Universal Robots PolyScope program: cubeDev.urp

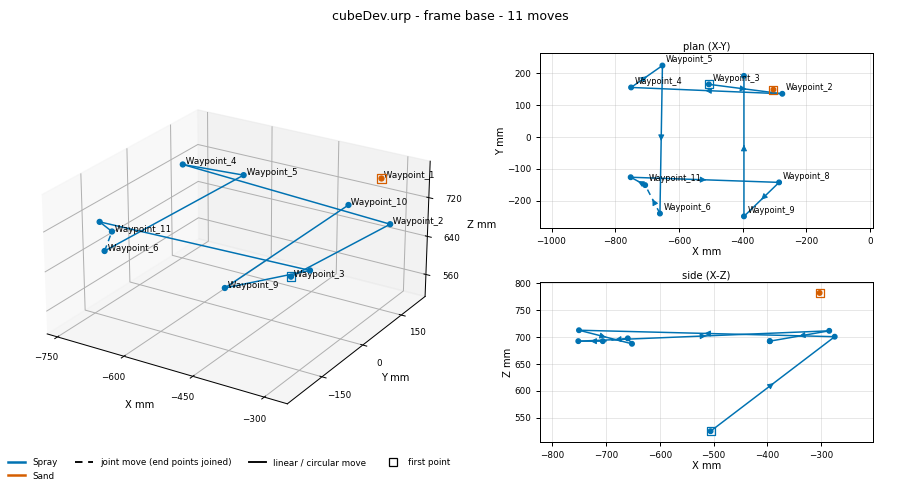
[picture p0: tool path of cubeDev.urp in frame base, 11 of 11 moves have a stored position in this frame; points joined in program order, loops and branches not executed]
Program cubeDev (installation=CubeDev directory=/programs/cube/archive createdIn=5.11.5.1010327 lastSavedIn=5.11.5.1010327 robotSerialNumber=20215500677)
Calibrated DH parameters: a=[0.000204, -0.239222, -0.391845, -0.000001, 0.000022, 0]; d=[0.162722, -355.808559, 353.37206, 2.570385, 0.099741, 0.099629]; alpha=[1.571124, 0.000988, 0.008295, 1.568963, -1.570303, 0]; deltaTheta=[0, -0.973091, 7.204745, 0.05153, 0, 0]
Robot Program (runOnlyOnce=false)
  Wait Sleep waitTime=0.01
SuppressedNode
  SubProgram LoadCube (keepSynchronizedWithDisk=false)
    Placeholder
Event  expression=digital_in[1]≟ True
  Call Spray
Event  expression=digital_in[2]≟ True
  Call Sand
  Call Sand
  Call Spray
  Call Spray
SubProgram -> Spray
SubProgram -> Sand
SubProgram Spray (keepSynchronizedWithDisk=false)
  Folder Spray
    Set NoAction tcp=SprayTCP
    MoveJ speed 60 deg/s, acceleration 80 deg/s^2 (useActiveTCP=false) tcp=SprayTCP; feature=Point_1
      Waypoint Waypoint_3: TCP in base x=-505.62 y=165.915 z=525.298 mm, rx=0.0993 ry=-0.0435 rz=1.9059 rad; joints [-54.164, 17.251, -106.459, 193.396, -48.457, -111.111] deg; TCP offset x=-60.833 y=-97.548 z=92.018 mm, rx=0.1226 ry=1.1769 rz=2.8697 rad; feature pose in base x=-342.399 y=157.897 z=730.093 mm, rx=-0.0205 ry=0.0193 rz=-1.2285 rad
    MoveL speed 180 mm/s, acceleration 1200 mm/s^2 (useActiveTCP=false) tcp=SprayTCP; feature=Point_1
      Waypoint Waypoint_2: TCP in base x=-275 y=136.265 z=700.836 mm, rx=0.7212 ry=-1.4137 rz=-0.8052 rad; joints [-53.492, 14.405, -127.134, 249.802, -70.84, -296.686] deg; TCP offset x=-60.833 y=-97.548 z=92.018 mm, rx=0.1226 ry=1.1769 rz=2.8697 rad; feature pose in base x=-342 y=157.897 z=730.093 mm, rx=-0.0205 ry=0.0193 rz=-1.2285 rad
      Set DigitalOutput pin=digital_out[5]; digitalValue=1
      Waypoint Waypoint_4: TCP in base x=-750 y=156.168 z=712.844 mm, rx=0.688 ry=-1.5401 rz=-0.8386 rad; joints [-18.358, -4.09, -33.202, 181.355, -101.612, -323.343] deg; TCP offset x=-60.833 y=-97.548 z=92.018 mm, rx=0.1226 ry=1.1769 rz=2.8697 rad
      Set DigitalOutput pin=digital_out[5]; digitalValue=0
      Waypoint Waypoint_5: TCP in base x=-651.58 y=225 z=687.663 mm, rx=1.4621 ry=-0.6099 rz=0.4016 rad; joints [-38.029, -10.685, -28.946, 126.451, -36.944, -216.931] deg; TCP offset x=-60.833 y=-97.548 z=92.018 mm, rx=0.1226 ry=1.1769 rz=2.8697 rad
      Set DigitalOutput pin=digital_out[5]; digitalValue=1
      Waypoint Waypoint_6: motionParameters(blendRadius=0.05); TCP in base x=-659.395 y=-239.888 z=697.768 mm, rx=1.4702 ry=-0.6913 rz=0.3254 rad; joints [5.108, 6.742, -60.072, 189.23, -54.458, -282.686] deg; TCP offset x=-60.833 y=-97.548 z=92.018 mm, rx=0.1226 ry=1.1769 rz=2.8697 rad
      Set DigitalOutput pin=digital_out[5]; digitalValue=0
    MoveJ speed 60 deg/s, acceleration 80 deg/s^2 (useActiveTCP=true positionType=JointAngles) feature=Base
      Waypoint Waypoint_11: TCP in base x=-705.785 y=-150.622 z=692.546 mm, rx=1.6603 ry=0.7065 rz=1.6076 rad; joints [-4.649, 6.051, -55.354, 271.275, 66.825, -330.102] deg
    MoveL speed 180 mm/s, acceleration 1200 mm/s^2 (useActiveTCP=false) tcp=SprayTCP; feature=Point_1
      Waypoint Waypoint_7: TCP in base x=-751.297 y=-125.892 z=692.562 mm, rx=1.6603 ry=0.7065 rz=1.6076 rad; joints [-6.168, 0.36, -40.894, 262.103, 67.957, -329.078] deg; feature pose in base x=-342 y=157.897 z=730.093 mm, rx=-0.0205 ry=0.0193 rz=-1.2285 rad
      Set DigitalOutput pin=digital_out[5]; digitalValue=1
      Waypoint Waypoint_8: TCP in base x=-285.147 y=-142.046 z=711.749 mm, rx=1.697 ry=0.7193 rz=1.5862 rad; joints [-12.195, 12.334, -126.012, 331.601, 72.274, -324.43] deg
      Set DigitalOutput pin=digital_out[5]; digitalValue=0
      Waypoint Waypoint_9: TCP in base x=-395.485 y=-248.751 z=692.565 mm, rx=-0.7915 ry=-1.8187 rz=-1.9759 rad; joints [17.792, 18.196, -97.975, 302.815, 116.578, -287.666] deg; feature pose in base x=-342.399 y=157.897 z=730.093 mm, rx=-0.0205 ry=0.0193 rz=-1.2285 rad
      Set DigitalOutput pin=digital_out[5]; digitalValue=1
      Waypoint Waypoint_10: TCP in base x=-395.529 y=192.479 z=692.53 mm, rx=-0.7913 ry=-1.8188 rz=-1.976 rad; joints [-32.817, 10.314, -105.902, 358.948, 141.949, -228.53] deg
      Set DigitalOutput pin=digital_out[5]; digitalValue=0
      MoveDirectionNode (selectedDirection=ZMinus) feature=Base
        Until DISTANCE (allowActions=false deceleration=3 distanceNodeType=STOP) Distance=0.05; motionParameters(blendRadius=0)
    SuppressedNode
      MoveJ speed 60 deg/s, acceleration 80 deg/s^2 (useActiveTCP=false) tcp=SandTCP; feature=Point_1
        Waypoint Waypoint_1: TCP in base x=-302.96 y=149.412 z=782.123 mm, rx=0 ry=0.0001 rz=-1.2192 rad; joints [-61.237, 0.512, -98.748, 196.199, -45.53, -101.275] deg; TCP offset x=3.18 y=114.64 z=98.2 mm, rx=-0.7854 ry=0 rz=0 rad; feature pose in base x=-302.957 y=149.397 z=782.11 mm, rx=0.0001 ry=0.0001 rz=-1.2192 rad
SubProgram Sand (keepSynchronizedWithDisk=false)
  Folder Sand
    MoveJ speed 60 deg/s, acceleration 80 deg/s^2 (useActiveTCP=false) tcp=SandTCP; feature=Point_1
      Waypoint Waypoint_1: TCP in base x=-302.96 y=149.412 z=782.123 mm, rx=0 ry=0.0001 rz=-1.2192 rad; joints [-61.237, 0.512, -98.748, 196.199, -45.53, -101.275] deg
    Wait Sleep waitTime=1
    MoveL speed 10 mm/s, acceleration 1200 mm/s^2 (useActiveTCP=true) feature=Base
      MoveDirectionNode (selectedDirection=ZPlus)
        Until TOOL_CONTACT_DETECTION (allowActions=false retraction=0 decelerationAcceleration=3 decelerationAngularAcceleration=34.906585)
    URCap Finishing Tool Control (Robotiq_Copilot, Robotiq Inc.) dataModel(ToolOutputNameKey=SanderOn, HackTriggeringContributionIsDefinedMethodKey=true)
    Force Simple feature=Base; selection=[0, 0, 1, 0, 0, 0]; wrench=[0, 0, 10, 0, 0, 0]; limitsForce=[0.15, 0.15, 0.15, 1.047198, 1.047198, 1.047198]; limitsMotion=[0.1, 0.1, 0.1, 0.349066, 0.349066, 0.349066]
      URCap Path Generator (Robotiq_Copilot, Robotiq Inc.) dataModel(pathOptionsTypeKey=TOOL_ON_ROBOT, PathTypeKey=FOUR_POINTS_HORIZONTAL, coverageModeKey=PERIMETER_ONLY, DimensionWidthTypeKey=FIXED, WaypointPoseKey1=[-0.302944, 0.149396, 0.782128, 1.50244E-5, 1.00412E-4, -1.21921], WaypointJointPositionsKey1=[-1.068778060252626, 0.008978874628797762, -1.7234921485718004, 3.4243521278056126, -0.7946231922406994, -1.767570591813545], WaypointPoseKey2=[-0.279518, -0.201261, 0.782103, 7.9768E-6, -3.58155E-5, -1.21905], WaypointJointPositionsKey2=[0.18023730066366817, 0.12175598563927537, -1.9454914874815659, 4.17217376502618, -1.4427139232998378, -3.0128294190106644], WaypointPoseKey3=[-0.644944, 0.149425, 0.782044, 1.44123E-5, -4.95705E-5, -1.21918], WaypointJointPositionsKey3=[-0.5050143034254404, -0.124510623031437, -0.715876541542217, 2.984549966298414, -1.008120014303917, -2.444335638266236], WaypointPoseKey4=[-0.6517, -0.201216, 0.782084, -6.15686E-7, -5.50915E-5, -1.21919], WaypointJointPositionsKey4=[0.07167613269606532, -0.07778302743568233, -0.7816102091272725, 3.1939898196044685, -1.3732669648021716, -2.9296232398659576], relativePathKey=true, selectedFeatureNameKey=Point_1, OriginalFeatureAsArrayKey=[-0.3029570133244077, 0.1493967343976849, 0.7821098019170267, 6.631708170368006E-5, 8.682855188236906E-5, -1.2191890682989344], offsetTypeKey=Relative to feature, PerimeterSpeedKey=100, urcapVersion=1.22.1); state(isChildrenLocked=true)
        URCap Point (Robotiq_Copilot, Robotiq Inc.) dataModel(pose=[-0.302944, 0.149396, 0.782128, 1.50244E-5, 1.00412E-4, -1.21921], joint_positions=[-1.068778060252626, 0.008978874628797762, -1.7234921485718004, 3.4243521278056126, -0.7946231922406994, -1.767570591813545])
        URCap Point (Robotiq_Copilot, Robotiq Inc.) dataModel(pose=[-0.279518, -0.201261, 0.782103, 7.9768E-6, -3.58155E-5, -1.21905], joint_positions=[0.18023730066366817, 0.12175598563927537, -1.9454914874815659, 4.17217376502618, -1.4427139232998378, -3.0128294190106644])
        URCap Point (Robotiq_Copilot, Robotiq Inc.) dataModel(pose=[-0.644944, 0.149425, 0.782044, 1.44123E-5, -4.95705E-5, -1.21918], joint_positions=[-0.5050143034254404, -0.124510623031437, -0.715876541542217, 2.984549966298414, -1.008120014303917, -2.444335638266236])
        URCap Point (Robotiq_Copilot, Robotiq Inc.) dataModel(pose=[-0.6517, -0.201216, 0.782084, -6.15686E-7, -5.50915E-5, -1.21919], joint_positions=[0.07167613269606532, -0.07778302743568233, -0.7816102091272725, 3.1939898196044685, -1.3732669648021716, -2.9296232398659576])
    URCap Finishing Tool Control (Robotiq_Copilot, Robotiq Inc.) dataModel(ToolOutputNameKey=SanderOn, HackTriggeringContributionIsDefinedMethodKey=true, FinishingToolStateKey=false)
    MoveL speed 250 mm/s, acceleration 1200 mm/s^2 (useActiveTCP=true) feature=Base
      MoveDirectionNode (selectedDirection=ZMinus) feature=Base
        Until DISTANCE (allowActions=false deceleration=3 distanceNodeType=STOP) Distance=0.075; motionParameters(blendRadius=0)
